FUNCTION_BLOCK IN_BOOL (* Boolean Input Checkbox *)
  (* Standard: 61499-1; Function: HMI; Type: BOOL input; Description: Checkbox *)
  (* Version 0.2, 2004-06-08, JHC, Rockwell Automation, Corrected documentation (no inhibitions). *)
  (* Version 0.1, 2002-05-03, JHC, Rockwell Automation, Made QI initial value =true. *)
  (* Version 0.0, 2001-03-08, JHC, Rockwell Automation, First XML version *)
  (* Compiler header: package fb.rt.awt; import java.awt.*; import java.awt.event.*; *)
  (* Compiler classdef: public class IN_BOOL extends FBInstance implements ItemListener *)
  (* Compiler Java IBM VisualAge 3.0 *)
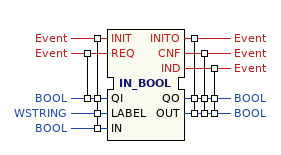
  EVENT_INPUT
    INIT WITH QI, LABEL, IN; (* Initialization *)
    REQ WITH QI; (* Request *)
  END_EVENT
  EVENT_OUTPUT
    INITO WITH QO, OUT; (* Initialization Confirm *)
    CNF WITH QO, OUT; (* Service Confirmation *)
    IND WITH QO, OUT; (* User clicked Checkbox *)
  END_EVENT
  VAR_INPUT
    QI : BOOL := true; (* Event qualifier *)
    LABEL : WSTRING; (* Label *)
    IN : BOOL; (* Initial value *)
  END_VAR
  VAR_OUTPUT
    QO : BOOL; (* Event qualifier *)
    OUT : BOOL; (* Output data *)
  END_VAR
  SERVICE IN_BOOL/Checkbox
    SEQUENCE normal_initialization
      IN_BOOL.INIT+(LABEL,IN) -> Checkbox.setLabel(LABEL) -> Checkbox.setState(IN) -> IN_BOOL.INITO+();
    END_SEQUENCE
    SEQUENCE initialization_inhibited
      IN_BOOL.INIT-() -> IN_BOOL.INITO-();
    END_SEQUENCE
    SEQUENCE data_read
      IN_BOOL.REQ+() -> Checkbox.getState() -> IN_BOOL.CNF+(OUT);
    END_SEQUENCE
    SEQUENCE user_input
      Checkbox.itemStateChanged() -> IN_BOOL.IND+(OUT);
    END_SEQUENCE
  END_SERVICE
END_FUNCTION_BLOCK
